// TwinCAT 3 PLC project PLC
// ProgramVersion: 3.1.4026.13
// libraries:
//   Tc2_Standard, * (Beckhoff Automation GmbH)
//   Tc2_System, * (Beckhoff Automation GmbH)
// project tree:
//   / PlcTask.TcTTO
//   POUs/ FB_Derivator.TcPOU, G_Init.TcGVL (not stored), MAIN.TcPOU
// real-time tasks:
//   TASK PlcTask: cycle T#10ms, priority 20, ADS port 350

CONFIGURATION PLC
    RESOURCE PLC ON TwinCAT3
        TASK PlcTask(INTERVAL := T#10ms, PRIORITY := 20);
        PROGRAM MAIN WITH PlcTask : MAIN;
    END_RESOURCE
END_CONFIGURATION

// ---- POUs/MAIN.TcPOU
PROGRAM MAIN
VAR
	fTimeStep : LREAL := 0.01;
	fTime : LREAL;
	fValue : LREAL;
	fbDerivator : FB_Derivator;
	bEnable : BOOL;
END_VAR

fTime := fTime + fTimeStep;

fbDerivator(
	ssMethodType := BOOL_TO_SINT(bEnable),
	fSignal := fTime,
	fSignalDerivative => fValue
	
);

END_PROGRAM

// ---- POUs/FB_Derivator.TcPOU
FUNCTION_BLOCK FB_Derivator
VAR_INPUT
	ssMethodType		: SINT;
	fSignal				: LREAL;
END_VAR
VAR_OUTPUT
	fSignalDerivative	: LREAL;
END_VAR
VAR
	rtb_TSamp			: LREAL;
	UD_DSTATE			: LREAL;
END_VAR



CASE ssMethodType OF
    SS_INITIALIZE: 
        (* SystemInitialize for Atomic SubSystem: '<Root>/Derivator' *)
        (* InitializeConditions for UnitDelay: '<S2>/UD'
         *
         * Block description for '<S2>/UD':
         *  
         *  Store in Global RAM *)
        UD_DSTATE := 0.0;
        (* End of SystemInitialize for SubSystem: '<Root>/Derivator' *)
    SS_STEP: 
        (* Outputs for Atomic SubSystem: '<Root>/Derivator' *)
        (* SampleTimeMath: '<S2>/TSamp'
         *
         * About '<S2>/TSamp':
         *  y = u * K where K = 1 / ( w * Ts )
         *   *)
        rtb_TSamp := fSignal * 100.0;
        (* Outport: '<Root>/fSignalDerivative' incorporates:
         *  Sum: '<S2>/Diff'
         *  UnitDelay: '<S2>/UD'
         *
         * Block description for '<S2>/Diff':
         *  
         *  Add in CPU
         *
         * Block description for '<S2>/UD':
         *  
         *  Store in Global RAM *)
        fSignalDerivative := rtb_TSamp - UD_DSTATE;
        (* Update for UnitDelay: '<S2>/UD'
         *
         * Block description for '<S2>/UD':
         *  
         *  Store in Global RAM *)
        UD_DSTATE := rtb_TSamp;
        (* End of Outputs for SubSystem: '<Root>/Derivator' *)
END_CASE;

END_FUNCTION_BLOCK
